(* IEC 61131-3 sources: POMIRTS_lab3/AS/Library_2/spooler, 3 files *)

(* ---- spooler.typ ---- *)
TYPE

END_TYPE

(* ---- spooler.fun ---- *)
{REDUND_ERROR} FUNCTION_BLOCK SPExUpData
	VAR_INPUT
		enable	:BOOL;
		pMode	:UDINT;
		pDevice	:UDINT;
		pIP	:UDINT;
		pCPU	:UDINT;
		data_len	:UDINT;
	END_VAR
	VAR_OUTPUT
		status	:UINT;
	END_VAR
	VAR
		first	:USINT;
		komm	:UDINT;
		maxcount	:UDINT;
		count	:UDINT;
		sp_dest	:UDINT;
		sp_kommadr	:UDINT;
		sp_mode	:UDINT;
	END_VAR
END_FUNCTION_BLOCK
{REDUND_ERROR} FUNCTION_BLOCK SPExDownData
	VAR_INPUT
		enable	:BOOL;
		pMode	:UDINT;
		pDevice	:UDINT;
		pIP	:UDINT;
		pCPU	:UDINT;
		data_len	:UDINT;
	END_VAR
	VAR_OUTPUT
		status	:UINT;
	END_VAR
	VAR
		first	:USINT;
		komm	:UDINT;
		maxcount	:UDINT;
		count	:UDINT;
		sp_dest	:UDINT;
		sp_kommadr	:UDINT;
		sp_mode	:UDINT;
	END_VAR
END_FUNCTION_BLOCK
{REDUND_ERROR} FUNCTION_BLOCK SPExUpModule
	VAR_INPUT
		enable	:BOOL;
		pMode	:UDINT;
		pDevice	:UDINT;
		pName	:UDINT;
	END_VAR
	VAR_OUTPUT
		status	:UINT;
		pCPU	:UDINT;
		pData	:UDINT;
		module_len	:UDINT;
	END_VAR
	VAR
		first	:USINT;
		komm	:UDINT;
		moadr	:UDINT;
		s_laenge	:UDINT;
		maxcount	:UDINT;
		count	:UDINT;
		sp_dest	:UDINT;
		sp_kommadr	:UDINT;
		sp_mode	:UDINT;
	END_VAR
END_FUNCTION_BLOCK
{REDUND_ERROR} FUNCTION_BLOCK SPExDownModule
	VAR_INPUT
		enable	:BOOL;
		pMode	:UDINT;
		pDevice	:UDINT;
		pName	:UDINT;
	END_VAR
	VAR_OUTPUT
		status	:UINT;
	END_VAR
	VAR
		first	:USINT;
		komm	:UDINT;
		moadr	:UDINT;
		maxcount	:UDINT;
		count	:UDINT;
		sp_dest	:UDINT;
		sp_kommadr	:UDINT;
		sp_mode	:UDINT;
	END_VAR
END_FUNCTION_BLOCK
{REDUND_ERROR} FUNCTION_BLOCK SPTimeOut
	VAR_INPUT
		enable	:BOOL;
		timeout	:USINT;
	END_VAR
	VAR_OUTPUT
		status	:UINT;
	END_VAR
END_FUNCTION_BLOCK
{REDUND_ERROR} FUNCTION_BLOCK SPUpData
	VAR_INPUT
		enable	:BOOL;
		io_type	:USINT;
		master_no	:USINT;
		slave_no	:USINT;
		module_adr	:USINT;
		mode	:USINT;
		ip_adr	:UDINT;
		cpu_adr	:UDINT;
		data_len	:UDINT;
	END_VAR
	VAR_OUTPUT
		status	:UINT;
	END_VAR
	VAR
		first	:USINT;
		komm	:UDINT;
		maxcount	:UDINT;
		count	:UDINT;
		sp_dest	:UDINT;
		sp_kommadr	:UDINT;
	END_VAR
END_FUNCTION_BLOCK
{REDUND_ERROR} FUNCTION_BLOCK SPDownData
	VAR_INPUT
		enable	:BOOL;
		io_type	:USINT;
		master_no	:USINT;
		slave_no	:USINT;
		module_adr	:USINT;
		mode	:USINT;
		ip_adr	:UDINT;
		cpu_adr	:UDINT;
		data_len	:UDINT;
	END_VAR
	VAR_OUTPUT
		status	:UINT;
	END_VAR
	VAR
		first	:USINT;
		komm	:UDINT;
		maxcount	:UDINT;
		count	:UDINT;
		sp_dest	:UDINT;
		sp_kommadr	:UDINT;
	END_VAR
END_FUNCTION_BLOCK
{REDUND_ERROR} FUNCTION_BLOCK SPUpModule
	VAR_INPUT
		enable	:BOOL;
		io_type	:USINT;
		master_no	:USINT;
		slave_no	:USINT;
		module_adr	:USINT;
		mode	:USINT;
		pName	:UDINT;
	END_VAR
	VAR_OUTPUT
		status	:UINT;
		cpu_adr	:UDINT;
		data_adr	:UDINT;
		modullen	:UDINT;
	END_VAR
	VAR
		first	:USINT;
		komm	:UDINT;
		moadr	:UDINT;
		s_laenge	:UDINT;
		maxcount	:UDINT;
		count	:UDINT;
		sp_dest	:UDINT;
		sp_kommadr	:UDINT;
	END_VAR
END_FUNCTION_BLOCK
{REDUND_ERROR} FUNCTION_BLOCK SPDownModule
	VAR_INPUT
		enable	:BOOL;
		io_type	:USINT;
		master_no	:USINT;
		slave_no	:USINT;
		module_adr	:USINT;
		mode	:USINT;
		pName	:UDINT;
	END_VAR
	VAR_OUTPUT
		status	:UINT;
	END_VAR
	VAR
		first	:USINT;
		komm	:UDINT;
		moadr	:UDINT;
		maxcount	:UDINT;
		count	:UDINT;
		sp_dest	:UDINT;
		sp_kommadr	:UDINT;
	END_VAR
END_FUNCTION_BLOCK

(* ---- spooler.var ---- *)
VAR CONSTANT
	spERR_SPF_RESET		: UINT	:= 6699;
	spERR_SPOOL_IOIMAGE	: UINT	:= 6670;
	spERR_SPOOLER_WORKING	: UINT	:= 6666;
	spERR_LONG_IRBOOT	: UINT	:= 6662;
	spERR_NOMORE_SPOOL	: UINT	:= 6660;
	spERR_SSP_SLERROR	: UINT	:= 6657;
	spERR_SSP_SLREADY	: UINT	:= 6655;
	spERR_SSP_NORESPONSE	: UINT	:= 6650;
	spERR_SPOOL_SLAVE_NO	: UINT	:= 6641;
	spERR_SPOOL_MASTER_NO	: UINT	:= 6640;
	spERR_SPOOL_QUEUE	: UINT	:= 6638;
	spERR_SPOOL_MODULADR	: UINT	:= 6637;
	spERR_SPOOL_NOMORE_READ	: UINT	:= 6635;
	spERR_SPOOL_MAX_INIT	: UINT	:= 6632;
	spERR_SPOOL_RIOTIMEOUT	: UINT	:= 6631;
	spERR_SPOOL_REMOTE_ADR	: UINT	:= 6629;
	spERR_SPOOL_SYSBUS_ADR	: UINT	:= 6628;
	spERR_SPOOL_IOTYP	: UINT	:= 6627;
	spERR_MSP_NOTIMPL	: UINT	:= 6610;
	spIO_TYPE_2005_IO	: USINT	:= 1;
	spIO_TYPE_2005_RIO	: USINT	:= 3;
	spIO_TYPE_2010_IO	: USINT	:= 0;
	spIO_TYPE_2010_RIO	: USINT	:= 2;
	spMASTER_NO_BASIS	: USINT	:= 1;
	spSLAVE_NO_BASIS	: USINT	:= 0;
	spSLAVE_NO_EXP1	: USINT	:= 1;
	spSLAVE_NO_EXP2	: USINT	:= 2;
	spSLAVE_NO_EXP3	: USINT	:= 3;
	spSLAVE_NO_EXP4	: USINT	:= 4;
END_VAR
